// TwinCAT 3 PLC project mobject_events
// Title: mobject-events
// Company: mobject
// Author: mobject dev team
// ProjectVersion: 1.1.0
// ProgramVersion: 3.1.4023.0
// libraries:
//   Tc2_System, * (Beckhoff Automation GmbH)
//   mobject-disposable,1.1.1,mobject
// project tree:
//   EventEmitter/ EventEmitter.TcPOU
//   Interfaces/ I_Event.TcIO, I_EventEmitter.TcIO, I_EventHandler.TcIO, I_EventTarget.TcIO
//   _Internal/EventHandlerItem/ EventHandlerItem.TcPOU, EventHandlerItemOnceOnly.TcPOU, I_EventHandlerItem.TcIO

// ---- Interfaces/I_Event.TcIO
INTERFACE I_Event EXTENDS __SYSTEM.IQueryInterface

END_INTERFACE

// ---- Interfaces/I_EventEmitter.TcIO
INTERFACE I_EventEmitter EXTENDS __SYSTEM.IQueryInterface

METHOD PUBLIC OffEvent
VAR_INPUT
	EventName : T_MaxString;
	EventHandler : I_EventHandler;
END_VAR
END_METHOD

METHOD PUBLIC OnceEvent
VAR_INPUT
	EventName : T_MaxString;
	EventHandler : I_EventHandler;
END_VAR
END_METHOD

METHOD PUBLIC OnEvent
VAR_INPUT
	EventName : T_MaxString;
	EventHandler : I_EventHandler;
END_VAR
END_METHOD

END_INTERFACE

// ---- Interfaces/I_EventHandler.TcIO
INTERFACE I_EventHandler EXTENDS __SYSTEM.IQueryInterface

METHOD PUBLIC HandleEvent
VAR_INPUT
	Event : I_Event;
END_VAR
END_METHOD

END_INTERFACE

// ---- Interfaces/I_EventTarget.TcIO
INTERFACE I_EventTarget EXTENDS __SYSTEM.IQueryInterface

METHOD PUBLIC Emit
VAR_INPUT
	EventName : T_MaxString;
	Event : I_Event;
END_VAR
END_METHOD

END_INTERFACE

// ---- _Internal/EventHandlerItem/I_EventHandlerItem.TcIO
INTERFACE I_EventHandlerItem EXTENDS I_Disposable

METHOD PUBLIC Emit
VAR_INPUT
	EventName : T_MaxString;
	Event : I_Event;
END_VAR
END_METHOD

METHOD PUBLIC EqualTo : BOOL
VAR_INPUT
	Name : T_MaxString;
	Handler : I_EventHandler;
END_VAR
END_METHOD

PROPERTY PUBLIC Next : I_EventHandlerItem
GET
END_GET
SET
END_SET
END_PROPERTY

PROPERTY PUBLIC Previous : I_EventHandlerItem
GET
END_GET
SET
END_SET
END_PROPERTY

END_INTERFACE

// ---- EventEmitter/EventEmitter.TcPOU
{attribute 'linkalways'} 
{attribute 'no_explicit_call' := 'This FB is a CLASS and must be accessed using methods or properties'}
{attribute 'enable_dynamic_creation'}
FUNCTION_BLOCK EventEmitter EXTENDS Disposable IMPLEMENTS I_EventEmitter, I_EventTarget
VAR
	firstEventHandlerItem : I_EventHandlerItem;
END_VAR

METHOD PUBLIC Clear
VAR_INPUT
END_VAR
DisposeAllEventHandlerItems();
END_METHOD

METHOD PRIVATE DisposeAllEventHandlerItems
VAR_INPUT
END_VAR
WHILE firstEventHandlerItem <> 0 DO
	DisposeEventHandlerItem(firstEventHandlerItem);
END_WHILE
END_METHOD

METHOD PRIVATE DisposeEventHandlerItem
VAR_INPUT
	EventHandlerItem : I_EventHandlerItem;
END_VAR
RemoveEventHandlerItemFromCollection(EventHandlerItem);
EventHandlerItem.Dispose();
END_METHOD

METHOD PUBLIC Emit
VAR_INPUT
	EventName : T_MaxString;
	Event : I_Event;
END_VAR
VAR
	currentEventHandlerItem : I_EventHandlerItem;
END_VAR
currentEventHandlerItem := firstEventHandlerItem;

WHILE currentEventHandlerItem <> 0 DO
	currentEventHandlerItem.Emit(EventName, Event);
	currentEventHandlerItem := currentEventHandlerItem.Next;
END_WHILE
END_METHOD

METHOD FB_exit : BOOL
VAR_INPUT
	bInCopyCode : BOOL; // if TRUE, the exit method is called for exiting an instance that is copied afterwards (online change).
END_VAR
IF bInCopyCode THEN
	RETURN;
END_IF

DisposeAllEventHandlerItems();
END_METHOD

METHOD PRIVATE FindEventHandlerItem : I_EventHandlerItem
VAR_INPUT
	EventName : T_MaxString;
	EventHandler : I_EventHandler;
END_VAR
VAR
	currentEventHandlerItem : I_EventHandlerItem;
END_VAR
currentEventHandlerItem := firstEventHandlerItem;

WHILE currentEventHandlerItem <> 0 DO
	
	IF currentEventHandlerItem.EqualTo(EventName, EventHandler) THEN
		FindEventHandlerItem := currentEventHandlerItem; 
		RETURN;
	END_IF
	
	currentEventHandlerItem := currentEventHandlerItem.Next;

END_WHILE
END_METHOD

METHOD PRIVATE InsertEventHandlerItem
VAR_INPUT
	EventHandlerItem : I_EventHandlerItem;
END_VAR
VAR
	currentEventHandlerItem : I_EventHandlerItem;
END_VAR
IF firstEventHandlerItem = 0 THEN
	firstEventHandlerItem := EventHandlerItem;
	RETURN;
END_IF

currentEventHandlerItem := firstEventHandlerItem;

WHILE currentEventHandlerItem.next <> 0 DO
	currentEventHandlerItem := currentEventHandlerItem.next;
END_WHILE

currentEventHandlerItem.next := EventHandlerItem;
EventHandlerItem.previous := currentEventHandlerItem;
END_METHOD

METHOD PUBLIC OffEvent
VAR_INPUT
	EventName : T_MaxString;
	EventHandler : I_EventHandler;
END_VAR
VAR
	foundHandlerItem : I_EventHandlerItem;
END_VAR
foundHandlerItem := FindEventHandlerItem(EventName, EventHandler);

IF foundHandlerItem = 0 THEN
	RETURN;
END_IF

DisposeEventHandlerItem(foundHandlerItem);
END_METHOD

METHOD PUBLIC OnceEvent
VAR_INPUT
	EventName : T_MaxString;
	EventHandler : I_EventHandler;
END_VAR
VAR
	pEventHandlerItem : POINTER TO EventHandlerItemOnceOnly;
END_VAR
pEventHandlerItem := __NEW(EventHandlerItemOnceOnly(Name := EventName, Handler := EventHandler, Parent := THIS^));
InsertEventHandlerItem(pEventHandlerItem^);
END_METHOD

METHOD PUBLIC OnEvent
VAR_INPUT
	EventName : T_MaxString;
	EventHandler : I_EventHandler;
END_VAR
VAR
	pEventHandlerItem : POINTER TO EventHandlerItem;
END_VAR
pEventHandlerItem := __NEW(EventHandlerItem(Name :=EventName, Handler := EventHandler));
InsertEventHandlerItem(pEventHandlerItem^);
END_METHOD

METHOD PRIVATE RemoveEventHandlerItemFromCollection
VAR_INPUT
	EventHandlerItem : I_EventHandlerItem;
END_VAR
VAR
	previous : I_EventHandlerItem;
	next : I_EventHandlerItem;
END_VAR
IF EventHandlerItem = 0 THEN
	// nothing to remove
	RETURN;
END_IF

IF EventHandlerItem = firstEventHandlerItem AND EventHandlerItem.Next = 0 THEN 
	
	// the item was the only one in the list, as such you just set the first to zero
	firstEventHandlerItem := 0; 
	
ELSIF EventHandlerItem = firstEventHandlerItem THEN 
	
	// the item was the first in the list of many, so make the next item the first and remove 
	// it's "previous" as the first in the item does not have a previous
	firstEventHandlerItem := EventHandlerItem.next; 
	firstEventHandlerItem.Previous := 0;

ELSIF EventHandlerItem.Next <> 0 THEN
	
	// the item is mid list so link it's previous and next together 
	previous := EventHandlerItem.Previous;
	next := EventHandlerItem.Next;
	
	previous.Next := next;
	next.Previous := previous;
	
ELSE 
	
	// the item is at the end so only remove itself from the previous
	previous := EventHandlerItem.Previous;
	previous.Next := 0;

END_IF
END_METHOD

END_FUNCTION_BLOCK

// ---- _Internal/EventHandlerItem/EventHandlerItem.TcPOU
{attribute 'linkalways'} 
{attribute 'no_explicit_call' := 'This FB is a CLASS and must be accessed using methods or properties'}
{attribute 'enable_dynamic_creation'}
FUNCTION_BLOCK EventHandlerItem EXTENDS Disposable IMPLEMENTS I_EventHandlerItem
VAR
	name : T_MAXSTRING;
	handler : I_EventHandler;
	_next : I_EventHandlerItem;
	_previous : I_EventHandlerItem;
END_VAR

METHOD PUBLIC Emit
VAR_INPUT
	EventName : T_MaxString;
	Event : I_Event;
END_VAR
IF EventName <> name THEN
	RETURN;
END_IF

IF handler = 0 THEN
	RETURN;
END_IF

handler.HandleEvent(Event);
END_METHOD

METHOD PUBLIC EqualTo : BOOL
VAR_INPUT
	Name : T_MaxString;
	Handler : I_EventHandler;
END_VAR
IF THIS^.handler <> Handler THEN
	RETURN;
END_IF

IF THIS^.name <> Name THEN
	RETURN;
END_IF

EqualTo := TRUE;
END_METHOD

METHOD FB_init : BOOL
VAR_INPUT
	bInitRetains : BOOL; // if TRUE, the retain variables are initialized (warm start / cold start)
	bInCopyCode : BOOL;  // if TRUE, the instance afterwards gets moved into the copy code (online change)
	Name : T_MAXSTRING;
	Handler : I_EventHandler;
END_VAR
THIS^.name := Name;
THIS^.handler := Handler;
END_METHOD

PROPERTY PUBLIC Next : I_EventHandlerItem
GET
Next := _next;
END_GET
SET
_next := Next;
END_SET
END_PROPERTY

PROPERTY PUBLIC Previous : I_EventHandlerItem
GET
Previous := _previous;
END_GET
SET
_previous := Previous;
END_SET
END_PROPERTY

END_FUNCTION_BLOCK

// ---- _Internal/EventHandlerItem/EventHandlerItemOnceOnly.TcPOU
{attribute 'linkalways'} 
{attribute 'no_explicit_call' := 'This FB is a CLASS and must be accessed using methods or properties'}
{attribute 'enable_dynamic_creation'}
FUNCTION_BLOCK EventHandlerItemOnceOnly EXTENDS EventHandlerItem
VAR
	parent : I_EventEmitter;
END_VAR

METHOD PUBLIC Emit
VAR_INPUT
	EventName : T_MaxString;
	Event : I_Event;
END_VAR
SUPER^.Emit(EventName,Event);
parent.OffEvent(name,handler);
END_METHOD

METHOD FB_init : BOOL
VAR_INPUT
	bInitRetains : BOOL; // if TRUE, the retain variables are initialized (warm start / cold start)
	bInCopyCode : BOOL;  // if TRUE, the instance afterwards gets moved into the copy code (online change)
	Name : T_MAXSTRING;
	Handler : I_EventHandler;
	Parent : I_EventEmitter;
END_VAR
THIS^.parent := Parent;
END_METHOD

END_FUNCTION_BLOCK
